(* CODESYS project SignalGen.library
   Author: m.kleven@beckhoff.com
   Version: 0.0.3
   Description: Signal generator algorithms
   Title: SignalGen
   Placeholder: SignalGen
   Company: Beckhoff Automation LLC.

Project tree, tasks and I/O mapping:
  libraries: Tc2_System, * (Beckhoff Automation GmbH)
  Project Information/
    function F_GetCompany [ST]
    function F_GetTitle [ST]
    function F_GetVersion [ST]
  Version/
    global variables Global_Version
  data type E_SawtoothType
  function block FB_SawtoothGenerator [ST]
  function block FB_SinewaveGenerator [ST]
  function block FB_SquareWaveGenerator [ST]
*)

// E_SawtoothType
{attribute 'qualified_only'}
{attribute 'strict'}
{attribute 'to_string'}
TYPE E_SawtoothType  :
(
    Rising := 0,    // Rising sawtooth (ramp up)
    Falling := 1    // Falling sawtooth (ramp down)
);
END_TYPE

// Version/Global_Version
{attribute 'TcGenerated'}
{attribute 'no-analysis'}
{attribute 'linkalways'}
// This function has been automatically generated from the project information.
VAR_GLOBAL CONSTANT
	{attribute 'const_non_replaced'}
	stLibVersion_SignalGen : ST_LibVersion := (iMajor := 0, iMinor := 0, iBuild := 3, iRevision := 0, nFlags := 0, sVersion := '0.0.3');
END_VAR

// Project Information/F_GetCompany
// This function has been automatically generated from the project information.
{attribute 'signature_flag' := '1073741824'}
{attribute 'TcGenerated'}
{attribute 'no-analysis'}
FUNCTION F_GetCompany : WSTRING
VAR_INPUT
	
END_VAR

F_GetCompany := "Beckhoff Automation LLC.";

END_FUNCTION

// Project Information/F_GetTitle
// This function has been automatically generated from the project information.
{attribute 'signature_flag' := '1073741824'}
{attribute 'TcGenerated'}
{attribute 'no-analysis'}
FUNCTION F_GetTitle : WSTRING
VAR_INPUT
	
END_VAR

F_GetTitle := "SignalGen";

END_FUNCTION

// Project Information/F_GetVersion
// This function has been automatically generated from the project information.
{attribute 'signature_flag' := '1073741824'}
{attribute 'TcGenerated'}
{attribute 'no-analysis'}
FUNCTION F_GetVersion : ST_LibVersion
VAR_INPUT
	
END_VAR

F_GetVersion.iMajor := 0;
F_GetVersion.iMinor := 0;
F_GetVersion.iBuild := 3;
F_GetVersion.iRevision := 0;
F_GetVersion.sVersion := '0.0.3';
F_GetVersion.nFlags := 0;

END_FUNCTION

// FB_SawtoothGenerator
FUNCTION_BLOCK FB_SawtoothGenerator
VAR_INPUT
	Enable	  : BOOL;									 // Enable generator
	Frequency : LREAL		   := 1.0;					 // Frequency in Hz
	Amplitude : LREAL		   := 1.0;					 // Amplitude (peak to peak)
	Offset	  : LREAL		   := 0.0;					 // DC offset
	SawType	  : E_SawtoothType := E_SawtoothType.Rising; // Sawtooth type
END_VAR

VAR_OUTPUT
	Output : LREAL; // Sawtooth wave output
	Error  : BOOL; // Error flag
END_VAR

VAR
	TimeAccum : LREAL;			// Internal time accumulator
	Period	  : LREAL;			// Period in seconds
	CycleTime : LREAL := 0.001; // 1ms cycle time (adjust as needed)
	TaskIdx	  : DINT;
	FirstScan : BOOL := TRUE;
END_VAR

IF FirstScan THEN
	FirstScan := FALSE;
	TaskIdx	  := GETCURTASKINDEXEX();
	IF TaskIdx > 0 THEN
		CycleTime := TO_LREAL(TwinCAT_SystemInfoVarList._TaskInfo[TaskIdx].CycleTime)/ 10000000.0;;
	END_IF
END_IF

IF Enable THEN
	// Input validation
	IF Frequency <= 0.0 THEN
		Error  := TRUE;
		Output := Offset;
		RETURN;
	END_IF

	// Calculate period
	Period := 1.0 / Frequency;

	// Accumulate time
	TimeAccum := TimeAccum + CycleTime;

	// Reset time at end of period
	IF TimeAccum >= Period THEN
		TimeAccum := TimeAccum - Period;
	END_IF

	// Generate sawtooth wave based on type
	CASE SawType OF
		E_SawtoothType.Rising:
			// Rising sawtooth: starts at -amplitude/2, rises to +amplitude/2
			Output := (TimeAccum / Period) * Amplitude - (Amplitude / 2.0) + Offset;

		E_SawtoothType.Falling:
			// Falling sawtooth: starts at +amplitude/2, falls to -amplitude/2
			Output := ((Period - TimeAccum) / Period) * Amplitude - (Amplitude / 2.0) + Offset;
	END_CASE

	Error := FALSE;
ELSE
	TimeAccum := 0.0;
	Output	  := Offset;
	Error	  := FALSE;
END_IF

END_FUNCTION_BLOCK

// FB_SinewaveGenerator
FUNCTION_BLOCK FB_SinewaveGenerator
VAR_INPUT
	Enable	  : BOOL;		  // Enable generator
	Frequency : LREAL := 1.0; // Frequency in Hz
	Amplitude : LREAL := 1.0; // Amplitude
	Offset	  : LREAL := 0.0; // DC offset
	Phase	  : LREAL := 0.0; // Phase offset in degrees
END_VAR

VAR_OUTPUT
	Output : LREAL; // Sine wave output
	Error  : BOOL; // Error flag
END_VAR

VAR
	TimeAccum : LREAL;			// Internal time accumulator
	DeltaTime : LREAL;			// Delta time per cycle
	PhaseRad  : LREAL;			// Phase in radians
	CycleTime : LREAL := 0.001; // 1ms cycle time (adjust as needed)
	TaskIdx	  : DINT;
	FirstScan : BOOL := TRUE;
END_VAR

// Function block code
IF FirstScan THEN
	FirstScan := FALSE;
	TaskIdx	  := GETCURTASKINDEXEX();
	IF TaskIdx > 0 THEN
		CycleTime := TO_LREAL(TwinCAT_SystemInfoVarList._TaskInfo[TaskIdx].CycleTime)/ 10000000.0;;
	END_IF
END_IF

IF Enable THEN
	// Convert phase from degrees to radians
	PhaseRad := Phase * Tc2_System.PI / 180.0;

	// Calculate delta time increment
	DeltaTime := Frequency * 2.0 * Tc2_System.PI * CycleTime;

	// Accumulate time
	TimeAccum := TimeAccum + DeltaTime;

	// Wrap time to prevent overflow
	IF TimeAccum >= 2.0 * Tc2_System.PI THEN
		TimeAccum := TimeAccum - 2.0 * Tc2_System.PI;
	END_IF

	// Generate sine wave
	Output := Amplitude * SIN(TimeAccum + PhaseRad) + Offset;
	Error  := FALSE;
ELSE
	TimeAccum := 0.0;
	Output	  := Offset;
	Error	  := FALSE;
END_IF

END_FUNCTION_BLOCK

// FB_SquareWaveGenerator
FUNCTION_BLOCK FB_SquareWaveGenerator
VAR_INPUT
    Enable     : BOOL;         // Enable generator
    Frequency  : LREAL := 1.0; // Frequency in Hz
    Amplitude  : LREAL := 1.0; // Amplitude (peak to peak)
    Offset     : LREAL := 0.0; // DC offset
    DutyCycle  : LREAL := 50.0; // Duty cycle in percentage (0-100)
END_VAR

VAR_OUTPUT
    Output     : LREAL; // Square wave output
    DigitalOut : BOOL; // Boolean output
    Error      : BOOL; // Error flag
END_VAR

VAR
    TimeAccum  : LREAL; // Internal time accumulator
    Period     : LREAL; // Period in seconds
    OnTime     : LREAL; // On time duration
    State      : BOOL;  // Current state
    CycleTime  : LREAL := 0.001; // 1ms cycle time (adjust as needed)
    TaskIdx    : DINT;
    FirstScan  : BOOL := TRUE;
END_VAR

IF FirstScan THEN
    FirstScan := FALSE;
    TaskIdx := GETCURTASKINDEXEX();
    IF TaskIdx > 0 THEN
        CycleTime := TO_LREAL(TwinCAT_SystemInfoVarList._TaskInfo[TaskIdx].CycleTime)/ 10000000.0;;
    END_IF
END_IF

IF Enable THEN
    // Input validation
    IF Frequency <= 0.0 OR DutyCycle < 0.0 OR DutyCycle > 100.0 THEN
        Error := TRUE;
        Output := Offset;
        DigitalOut := FALSE;
        RETURN;
    END_IF
    
    // Calculate period and on time
    Period := 1.0 / Frequency;
    OnTime := Period * DutyCycle / 100.0;
    
    // Accumulate time
    TimeAccum := TimeAccum + CycleTime;
    
    // Reset time at end of period
    IF TimeAccum >= Period THEN
        TimeAccum := TimeAccum - Period;
    END_IF
    
    // Determine output state
    State := TimeAccum < OnTime;
    DigitalOut := State;
    
    // Generate square wave output
    IF State THEN
        Output := Amplitude / 2.0 + Offset;
    ELSE
        Output := -Amplitude / 2.0 + Offset;
    END_IF
    
    Error := FALSE;
ELSE
    TimeAccum := 0.0;
    Output := Offset;
    DigitalOut := FALSE;
    Error := FALSE;
END_IF

END_FUNCTION_BLOCK
